{attribute 'GeneratedUsingTerminal: EP7211-0035-0029'}
{attribute addProperty BoxType "EP7211-0035-0029"}
{attribute addProperty Id "ControlwordAT %Q*UINT2"}
{attribute addProperty CRC "4092675873"}
{attribute addProperty Size "2"}
TYPE DS402_Controlword_F3F14721 :
STRUCT
	{attribute addProperty Name "Controlword"}
	Controlword AT %Q* : UINT;
END_STRUCT
END_TYPE

(* stored: Version 1.2.0.0, ProductVersion 3.1.4024.9
   DUT DS402_Controlword_F3F14721: Id {273f9309-b4a9-4bec-a4e3-b598f126875b} *)
